Universal Robots URScript: 20241121_contact_test.script

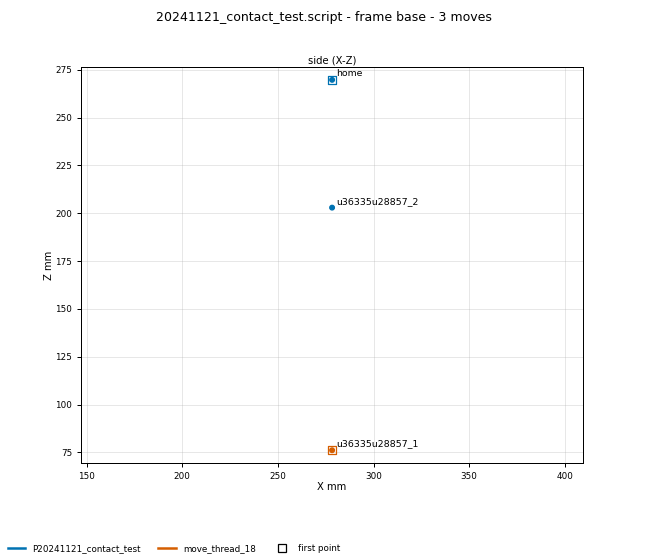
[picture p0: tool path of 20241121_contact_test.script in frame base, 3 of 3 moves have a stored position in this frame; points joined in program order, loops and branches not executed]
def P20241121_contact_test():
  global _hidden_verificationVariable=0
  set_target_payload(1.500000, [0.001000, -0.003000, 0.050000], [0.003026, 0.003026, 0.003026, 0.000000, 0.000000, 0.000000])
  set_tcp(p[-1.7E-4,0.0,0.19294999999999998,0.0,0.0,0.0])
  set_tool_communication(True, 115200, 0, 1, 1.5, 3.5)
  set_tool_output_mode(0)
  set_tool_digital_output_mode(0, 1)
  set_tool_digital_output_mode(1, 1)
  set_tool_voltage(24)
  set_standard_analog_input_domain(0, 1)
  set_standard_analog_input_domain(1, 1)
  set_tool_analog_input_domain(0, 1)
  set_tool_analog_input_domain(1, 1)
  set_analog_outputdomain(0, 1)
  set_analog_outputdomain(1, 0)
  set_input_actions_to_default()
  set_tool_digital_input_action(0, "freedrive")
  set_gravity([0.0, 0.0, 9.82])
  set_safety_mode_transition_hardness(0)
  global i_var_1=p[0.31, 0, 0, 0, 0, 0]
  global u24179u38754_1=p[0.0,0.0,0.0,0.0,0.0,0.0]
  global u24179u38754_2=p[0.2,0.6,0.4,-1.4839444017850547,-0.07419722008925289,-2.225916602677581]
  global u24179u38754_3=p[0.1459477485431481,-0.10308445883660293,0.13857682671027435,-0.008977024873201634,0.014216906208388691,-2.4400986907073663]
  global u28857_1=p[0.10203918836050063,-0.5259531579406657,0.376430278847906,-0.18768520041296463,-3.1325095402283982,-0.09669790600413578]
  global u28857_2=p[0.0665007526844362,-0.3872123180436422,0.638459113340625,-0.320095108678139,-2.6903368475934015,1.4700117755369673]
  global u30452u32447_1=p[0.0,0.0,0.0,0.0,0.0,0.0]
  step_count_b4d2483f_8893_49b8_936f_64b158deedd3 = 0.0
  thread Step_Counter_Thread_a2b80ebc_5de6_4f94_bd03_a8c00072d35d():
    while (True):
      step_count_b4d2483f_8893_49b8_936f_64b158deedd3 = step_count_b4d2483f_8893_49b8_936f_64b158deedd3 + 1.0
      sync()
    end
  end
  run Step_Counter_Thread_a2b80ebc_5de6_4f94_bd03_a8c00072d35d()
  global home_p=p[.278360590718, -.491587447341, .269714935010, -2.163959557712, -2.155629600597, -.000504384949]
  global home_q=[1.8672124147415161, -1.3750526917031785, 1.4028156439410608, -1.5219572123936196, -1.6108649412738245, 1.8757604360580444]
  global u36335u28857_1_p=p[.278354031362, -.491579900424, .076094230343, -2.285413173902, -2.155554113167, -.000000680795]
  global u36335u28857_1_q=[1.8457586765289307, -1.299463377600052, 1.8455475012408655, -2.1176282368102015, -1.571679417287008, 1.907263994216919]
  global u36335u28857_2_p=p[.278344002702, -.491572981319, .202918048913, -2.285367170671, -2.155524988368, -.000018936798]
  global u36335u28857_2_q=[1.8457670211791992, -1.4131920796683808, 1.6372054258929651, -1.7955056629576625, -1.5709870497332972, 1.9073389768600464]
  $ 23 "Thread_1"
  thread Thread_1():
    while (True):
      $ 24 "tmp≔p[0,0,0,0,0,0]"
      global tmp=p[0,0,0,0,0,0]
      $ 25 "循环"
      while (True):
        $ 26 "watchdog≔read_input_integer_register(0)"
        global watchdog=read_input_integer_register(0)
        $ 27 "脚本: pose_register.script"
        tmp[0]=read_input_float_register(0)
        tmp[1]=read_input_float_register(1)
        tmp[2]=read_input_float_register(2)
        tmp[3]=read_input_float_register(3)
        tmp[4]=read_input_float_register(4)
        tmp[5]=read_input_float_register(5)
        $ 28 "sync()"
        sync()
      end
    end
  end
  threadId_Thread_1 = run Thread_1()
  while (True):
    $ 2 "机器人程序"
    $ 3 "usb = rpc_factory('xmlrpc','http://192.168.1.3:9120/RPC2')"
    usb = rpc_factory("xmlrpc","http://192.168.1.3:9120/RPC2")
    $ 4 "弹出窗口: place check everything is ok!"
    popup("place check everything is ok!", "消息", False, False, blocking=True)
    $ 5 "write_output_integer_register(0,1)"
    write_output_integer_register(0,1)
    $ 7 "MoveJ"
    $ 8 "home" "breakAfter"
    movej(get_inverse_kin(home_p, qnear=home_q), a=1.3962634015954636, v=1.0471975511965976)
    $ 9 "usb.open()"
    usb.open()
    $ 10 "弹出窗口: close"
    popup("close", "消息", False, False, blocking=True)
    $ 11 "usb.adaptiveClose()"
    usb.adaptiveClose()
    $ 13 "等待: 2.0"
    sleep(2.0)
    $ 15 "循环"
    while (True):
      $ 16 "usb.enableSlipDetector()"
      usb.enableSlipDetector()
      $ 17 "MoveL"
      $ 18 "路点_1" "breakAfter"
      global move_thread_flag_18=0
      thread move_thread_18():
        enter_critical
        move_thread_flag_18 = 1
        movel(u36335u28857_1_p, a=0.5, v=0.1)
        move_thread_flag_18 = 2
        exit_critical
      end
      move_thread_flag_18 = 0
      move_thread_han_18 = run move_thread_18()
      while (True):
        if (tmp[0]>1):
          kill move_thread_han_18
          stopl(35.0)
          $ 19 "Until (expression)"
          break
        end
        sleep(1.0E-10)
        if (move_thread_flag_18 > 1):
          join move_thread_han_18
          break
        end
        sync()
      end
      $ 20 "等待: 2.0"
      sleep(2.0)
      $ 21 "usb.disEnableSlipDetector()"
      usb.disEnableSlipDetector()
      $ 22 "路点_2" "breakAfter"
      movel(u36335u28857_2_p, a=0.5, v=0.1)
    end
  end
end
